REGION Network 53: Step[910] : Transfer PP Right X/Z-Axis Weight Check Pos
   RUNG wire#powerrail
      { S7_Templates := "SrcType := DInt" } EQ_Contact(in1 := "Unit1.Em5.ControlNodes".transferPnPRight.sequence.status.currentStep, in2 := #JOB_9_STEP_10)
      Contact( "Unit1.Em5.ControlNodes".transferPnPRight.sequence.status.seqActive )
      wire#w1
      I_Contact( "Unit1.Em5.ControlNodes".cm.softcam.transferPnPRightAxisX.pos04_weightCheck.inPos )
      wire#w2
      Coil( "Unit1.Em5.ControlNodes".transferPnPRight."step".action1[910] )
   END_RUNG
   RUNG wire#w1
      I_Contact( "Unit1.Em5.ControlNodes".cm.softcam.transferPnPRightAxisZ.pos04_weightCheck1.inPos )
   END_RUNG wire#w2
   RUNG wire#w1
      Contact( "Unit1.Em5.ControlNodes".cm.softcam.transferPnPRightAxisX.pos04_weightCheck.inPos )
      Contact( "Unit1.Em5.ControlNodes".cm.softcam.transferPnPRightAxisZ.pos04_weightCheck1.inPos )
      Coil( "Unit1.Em5.ControlNodes".transferPnPRight."step".transition1[910] )
   END_RUNG
   RUNG wire#w1
      Contact( "Unit1.Em5.ControlNodes".transferPnPRight."step".transition1[910] )
      { S7_Templates := "time_type := Time" } #statTonTime[910].TON(pt := T#100ms, et =>)
      Move(in := #JOB_9_STEP_30, out1 => "Unit1.Em5.ControlNodes".transferPnPRight.sequence.status.nextStep)
   END_RUNG
   // the same network as SCL:
   #_w1 := ("Unit1.Em5.ControlNodes".transferPnPRight.sequence.status.currentStep = #JOB_9_STEP_10) AND "Unit1.Em5.ControlNodes".transferPnPRight.sequence.status.seqActive;
   "Unit1.Em5.ControlNodes".transferPnPRight."step".action1[910] := #_w1 AND (NOT "Unit1.Em5.ControlNodes".cm.softcam.transferPnPRightAxisX.pos04_weightCheck.inPos OR NOT "Unit1.Em5.ControlNodes".cm.softcam.transferPnPRightAxisZ.pos04_weightCheck1.inPos);
   "Unit1.Em5.ControlNodes".transferPnPRight."step".transition1[910] := #_w1 AND "Unit1.Em5.ControlNodes".cm.softcam.transferPnPRightAxisX.pos04_weightCheck.inPos AND "Unit1.Em5.ControlNodes".cm.softcam.transferPnPRightAxisZ.pos04_weightCheck1.inPos;
   #statTonTime[910].TON(IN := #_w1 AND "Unit1.Em5.ControlNodes".transferPnPRight."step".transition1[910],
                         PT := T#100ms);
   IF #statTonTime[910].Q THEN
       "Unit1.Em5.ControlNodes".transferPnPRight.sequence.status.nextStep := #JOB_9_STEP_30;
   END_IF;
END_REGION

REGION Network 54: Step[930] : Transfer PP Right Y-Axis Weight Check Pos
   RUNG wire#powerrail
      { S7_Templates := "SrcType := DInt" } EQ_Contact(in1 := "Unit1.Em5.ControlNodes".transferPnPRight.sequence.status.currentStep, in2 := #JOB_9_STEP_30)
      Contact( "Unit1.Em5.ControlNodes".transferPnPRight.sequence.status.seqActive )
      wire#w1
      I_Contact( "Unit1.Em5.ControlNodes".cm.softcam.transferPnPRightAxisY.pos04_weightCheck.inPos )
      Coil( "Unit1.Em5.ControlNodes".transferPnPRight."step".action1[930] )
   END_RUNG
   RUNG wire#w1
      Contact( "Unit1.Em5.ControlNodes".cm.softcam.transferPnPRightAxisY.pos04_weightCheck.inPos )
      Coil( "Unit1.Em5.ControlNodes".transferPnPRight."step".transition1[930] )
   END_RUNG
   RUNG wire#w1
      Contact( "Unit1.Em5.ControlNodes".transferPnPRight."step".transition1[930] )
      { S7_Templates := "time_type := Time" } #statTonTime[930].TON(pt := T#100ms, et =>)
      Move(in := #JOB_9_STEP_31, out1 => "Unit1.Em5.ControlNodes".transferPnPRight.sequence.status.nextStep)
   END_RUNG
   // the same network as SCL:
   #_w1 := ("Unit1.Em5.ControlNodes".transferPnPRight.sequence.status.currentStep = #JOB_9_STEP_30) AND "Unit1.Em5.ControlNodes".transferPnPRight.sequence.status.seqActive;
   "Unit1.Em5.ControlNodes".transferPnPRight."step".action1[930] := #_w1 AND NOT "Unit1.Em5.ControlNodes".cm.softcam.transferPnPRightAxisY.pos04_weightCheck.inPos;
   "Unit1.Em5.ControlNodes".transferPnPRight."step".transition1[930] := #_w1 AND "Unit1.Em5.ControlNodes".cm.softcam.transferPnPRightAxisY.pos04_weightCheck.inPos;
   #statTonTime[930].TON(IN := #_w1 AND "Unit1.Em5.ControlNodes".transferPnPRight."step".transition1[930],
                         PT := T#100ms);
   IF #statTonTime[930].Q THEN
       "Unit1.Em5.ControlNodes".transferPnPRight.sequence.status.nextStep := #JOB_9_STEP_31;
   END_IF;
END_REGION

REGION Network 55: Step[931] : Transfer PP Right Z-Axis Weight Check Pos
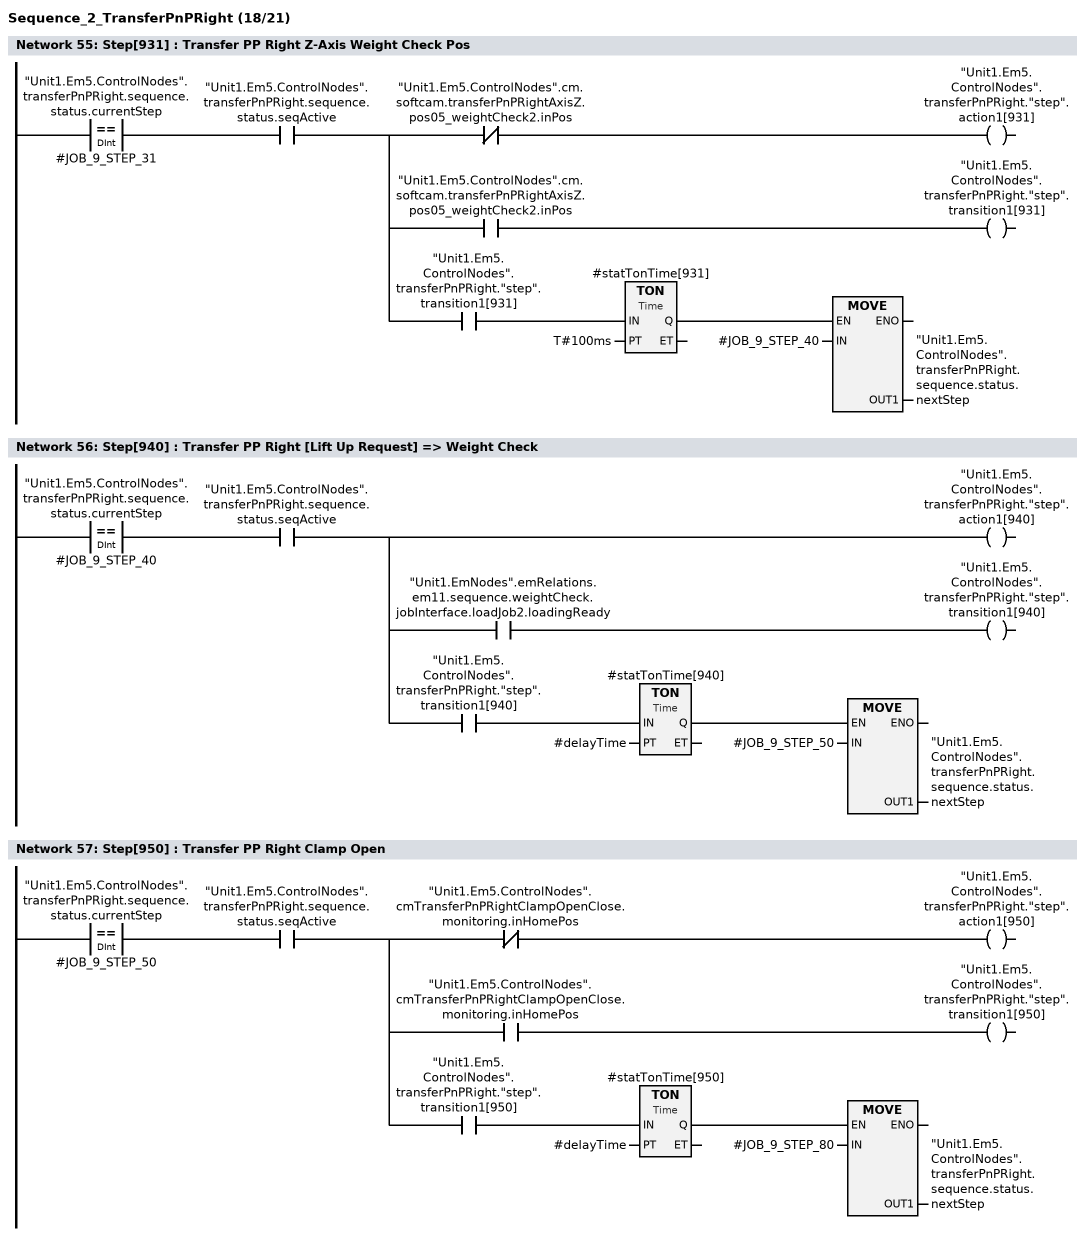
   RUNG wire#powerrail
      { S7_Templates := "SrcType := DInt" } EQ_Contact(in1 := "Unit1.Em5.ControlNodes".transferPnPRight.sequence.status.currentStep, in2 := #JOB_9_STEP_31)
      Contact( "Unit1.Em5.ControlNodes".transferPnPRight.sequence.status.seqActive )
      wire#w1
      I_Contact( "Unit1.Em5.ControlNodes".cm.softcam.transferPnPRightAxisZ.pos05_weightCheck2.inPos )
      Coil( "Unit1.Em5.ControlNodes".transferPnPRight."step".action1[931] )
   END_RUNG
   RUNG wire#w1
      Contact( "Unit1.Em5.ControlNodes".cm.softcam.transferPnPRightAxisZ.pos05_weightCheck2.inPos )
      Coil( "Unit1.Em5.ControlNodes".transferPnPRight."step".transition1[931] )
   END_RUNG
   RUNG wire#w1
      Contact( "Unit1.Em5.ControlNodes".transferPnPRight."step".transition1[931] )
      { S7_Templates := "time_type := Time" } #statTonTime[931].TON(pt := T#100ms, et =>)
      Move(in := #JOB_9_STEP_40, out1 => "Unit1.Em5.ControlNodes".transferPnPRight.sequence.status.nextStep)
   END_RUNG
   // the same network as SCL:
   #_w1 := ("Unit1.Em5.ControlNodes".transferPnPRight.sequence.status.currentStep = #JOB_9_STEP_31) AND "Unit1.Em5.ControlNodes".transferPnPRight.sequence.status.seqActive;
   "Unit1.Em5.ControlNodes".transferPnPRight."step".action1[931] := #_w1 AND NOT "Unit1.Em5.ControlNodes".cm.softcam.transferPnPRightAxisZ.pos05_weightCheck2.inPos;
   "Unit1.Em5.ControlNodes".transferPnPRight."step".transition1[931] := #_w1 AND "Unit1.Em5.ControlNodes".cm.softcam.transferPnPRightAxisZ.pos05_weightCheck2.inPos;
   #statTonTime[931].TON(IN := #_w1 AND "Unit1.Em5.ControlNodes".transferPnPRight."step".transition1[931],
                         PT := T#100ms);
   IF #statTonTime[931].Q THEN
       "Unit1.Em5.ControlNodes".transferPnPRight.sequence.status.nextStep := #JOB_9_STEP_40;
   END_IF;
END_REGION

REGION Network 56: Step[940] : Transfer PP Right [Lift Up Request] => Weight Check
   RUNG wire#powerrail
      { S7_Templates := "SrcType := DInt" } EQ_Contact(in1 := "Unit1.Em5.ControlNodes".transferPnPRight.sequence.status.currentStep, in2 := #JOB_9_STEP_40)
      Contact( "Unit1.Em5.ControlNodes".transferPnPRight.sequence.status.seqActive )
      wire#w1
      Coil( "Unit1.Em5.ControlNodes".transferPnPRight."step".action1[940] )
   END_RUNG
   RUNG wire#w1
      Contact( "Unit1.EmNodes".emRelations.em11.sequence.weightCheck.jobInterface.loadJob2.loadingReady )
      Coil( "Unit1.Em5.ControlNodes".transferPnPRight."step".transition1[940] )
   END_RUNG
   RUNG wire#w1
      Contact( "Unit1.Em5.ControlNodes".transferPnPRight."step".transition1[940] )
      { S7_Templates := "time_type := Time" } #statTonTime[940].TON(pt := #delayTime, et =>)
      Move(in := #JOB_9_STEP_50, out1 => "Unit1.Em5.ControlNodes".transferPnPRight.sequence.status.nextStep)
   END_RUNG
   // the same network as SCL:
   "Unit1.Em5.ControlNodes".transferPnPRight."step".action1[940] := ("Unit1.Em5.ControlNodes".transferPnPRight.sequence.status.currentStep = #JOB_9_STEP_40) AND "Unit1.Em5.ControlNodes".transferPnPRight.sequence.status.seqActive;
   "Unit1.Em5.ControlNodes".transferPnPRight."step".transition1[940] := ("Unit1.Em5.ControlNodes".transferPnPRight.sequence.status.currentStep = #JOB_9_STEP_40) AND "Unit1.Em5.ControlNodes".transferPnPRight.sequence.status.seqActive AND "Unit1.EmNodes".emRelations.em11.sequence.weightCheck.jobInterface.loadJob2.loadingReady;
   #statTonTime[940].TON(IN := ("Unit1.Em5.ControlNodes".transferPnPRight.sequence.status.currentStep = #JOB_9_STEP_40) AND "Unit1.Em5.ControlNodes".transferPnPRight.sequence.status.seqActive AND "Unit1.Em5.ControlNodes".transferPnPRight."step".transition1[940],
                         PT := #delayTime);
   IF #statTonTime[940].Q THEN
       "Unit1.Em5.ControlNodes".transferPnPRight.sequence.status.nextStep := #JOB_9_STEP_50;
   END_IF;
END_REGION

REGION Network 57: Step[950] : Transfer PP Right Clamp Open
   RUNG wire#powerrail
      { S7_Templates := "SrcType := DInt" } EQ_Contact(in1 := "Unit1.Em5.ControlNodes".transferPnPRight.sequence.status.currentStep, in2 := #JOB_9_STEP_50)
      Contact( "Unit1.Em5.ControlNodes".transferPnPRight.sequence.status.seqActive )
      wire#w1
      I_Contact( "Unit1.Em5.ControlNodes".cmTransferPnPRightClampOpenClose.monitoring.inHomePos )
      Coil( "Unit1.Em5.ControlNodes".transferPnPRight."step".action1[950] )
   END_RUNG
   RUNG wire#w1
      Contact( "Unit1.Em5.ControlNodes".cmTransferPnPRightClampOpenClose.monitoring.inHomePos )
      Coil( "Unit1.Em5.ControlNodes".transferPnPRight."step".transition1[950] )
   END_RUNG
   RUNG wire#w1
      Contact( "Unit1.Em5.ControlNodes".transferPnPRight."step".transition1[950] )
      { S7_Templates := "time_type := Time" } #statTonTime[950].TON(pt := #delayTime, et =>)
      Move(in := #JOB_9_STEP_80, out1 => "Unit1.Em5.ControlNodes".transferPnPRight.sequence.status.nextStep)
   END_RUNG
   // the same network as SCL:
   #_w1 := ("Unit1.Em5.ControlNodes".transferPnPRight.sequence.status.currentStep = #JOB_9_STEP_50) AND "Unit1.Em5.ControlNodes".transferPnPRight.sequence.status.seqActive;
   "Unit1.Em5.ControlNodes".transferPnPRight."step".action1[950] := #_w1 AND NOT "Unit1.Em5.ControlNodes".cmTransferPnPRightClampOpenClose.monitoring.inHomePos;
   "Unit1.Em5.ControlNodes".transferPnPRight."step".transition1[950] := #_w1 AND "Unit1.Em5.ControlNodes".cmTransferPnPRightClampOpenClose.monitoring.inHomePos;
   #statTonTime[950].TON(IN := #_w1 AND "Unit1.Em5.ControlNodes".transferPnPRight."step".transition1[950],
                         PT := #delayTime);
   IF #statTonTime[950].Q THEN
       "Unit1.Em5.ControlNodes".transferPnPRight.sequence.status.nextStep := #JOB_9_STEP_80;
   END_IF;
END_REGION

REGION Network 58: Step[980] : Transfer PP Right Y-Axis Wait Pos
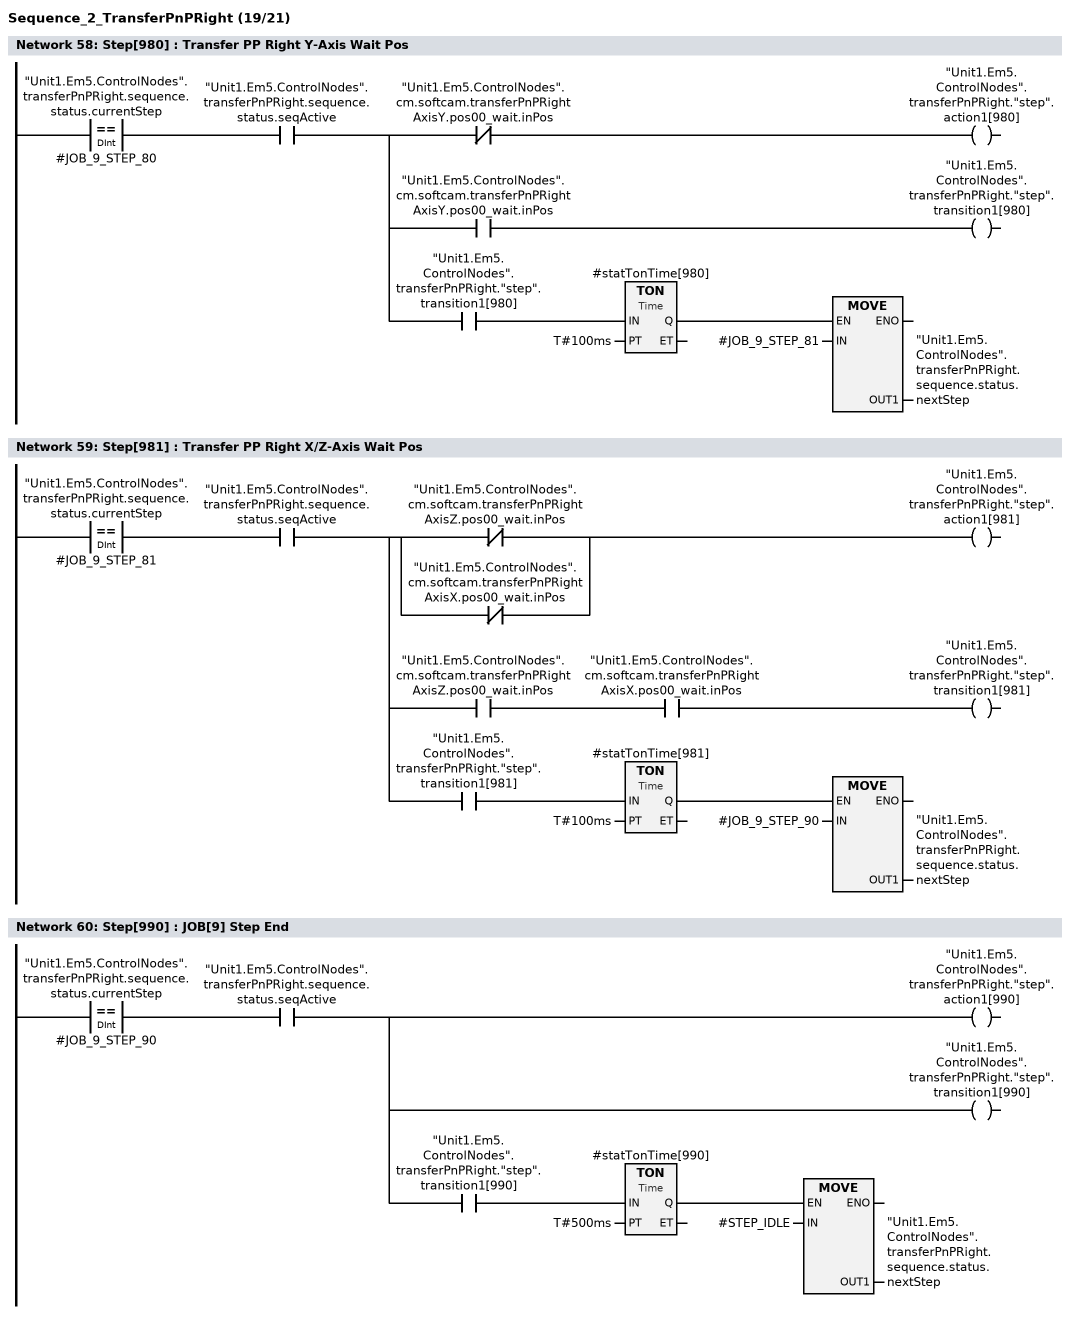
   RUNG wire#powerrail
      { S7_Templates := "SrcType := DInt" } EQ_Contact(in1 := "Unit1.Em5.ControlNodes".transferPnPRight.sequence.status.currentStep, in2 := #JOB_9_STEP_80)
      Contact( "Unit1.Em5.ControlNodes".transferPnPRight.sequence.status.seqActive )
      wire#w1
      I_Contact( "Unit1.Em5.ControlNodes".cm.softcam.transferPnPRightAxisY.pos00_wait.inPos )
      Coil( "Unit1.Em5.ControlNodes".transferPnPRight."step".action1[980] )
   END_RUNG
   RUNG wire#w1
      Contact( "Unit1.Em5.ControlNodes".cm.softcam.transferPnPRightAxisY.pos00_wait.inPos )
      Coil( "Unit1.Em5.ControlNodes".transferPnPRight."step".transition1[980] )
   END_RUNG
   RUNG wire#w1
      Contact( "Unit1.Em5.ControlNodes".transferPnPRight."step".transition1[980] )
      { S7_Templates := "time_type := Time" } #statTonTime[980].TON(pt := T#100ms, et =>)
      Move(in := #JOB_9_STEP_81, out1 => "Unit1.Em5.ControlNodes".transferPnPRight.sequence.status.nextStep)
   END_RUNG
   // the same network as SCL:
   #_w1 := ("Unit1.Em5.ControlNodes".transferPnPRight.sequence.status.currentStep = #JOB_9_STEP_80) AND "Unit1.Em5.ControlNodes".transferPnPRight.sequence.status.seqActive;
   "Unit1.Em5.ControlNodes".transferPnPRight."step".action1[980] := #_w1 AND NOT "Unit1.Em5.ControlNodes".cm.softcam.transferPnPRightAxisY.pos00_wait.inPos;
   "Unit1.Em5.ControlNodes".transferPnPRight."step".transition1[980] := #_w1 AND "Unit1.Em5.ControlNodes".cm.softcam.transferPnPRightAxisY.pos00_wait.inPos;
   #statTonTime[980].TON(IN := #_w1 AND "Unit1.Em5.ControlNodes".transferPnPRight."step".transition1[980],
                         PT := T#100ms);
   IF #statTonTime[980].Q THEN
       "Unit1.Em5.ControlNodes".transferPnPRight.sequence.status.nextStep := #JOB_9_STEP_81;
   END_IF;
END_REGION

REGION Network 59: Step[981] : Transfer PP Right X/Z-Axis Wait Pos
   RUNG wire#powerrail
      { S7_Templates := "SrcType := DInt" } EQ_Contact(in1 := "Unit1.Em5.ControlNodes".transferPnPRight.sequence.status.currentStep, in2 := #JOB_9_STEP_81)
      Contact( "Unit1.Em5.ControlNodes".transferPnPRight.sequence.status.seqActive )
      wire#w1
      I_Contact( "Unit1.Em5.ControlNodes".cm.softcam.transferPnPRightAxisZ.pos00_wait.inPos )
      wire#w2
      Coil( "Unit1.Em5.ControlNodes".transferPnPRight."step".action1[981] )
   END_RUNG
   RUNG wire#w1
      I_Contact( "Unit1.Em5.ControlNodes".cm.softcam.transferPnPRightAxisX.pos00_wait.inPos )
   END_RUNG wire#w2
   RUNG wire#w1
      Contact( "Unit1.Em5.ControlNodes".cm.softcam.transferPnPRightAxisZ.pos00_wait.inPos )
      Contact( "Unit1.Em5.ControlNodes".cm.softcam.transferPnPRightAxisX.pos00_wait.inPos )
      Coil( "Unit1.Em5.ControlNodes".transferPnPRight."step".transition1[981] )
   END_RUNG
   RUNG wire#w1
      Contact( "Unit1.Em5.ControlNodes".transferPnPRight."step".transition1[981] )
      { S7_Templates := "time_type := Time" } #statTonTime[981].TON(pt := T#100ms, et =>)
      Move(in := #JOB_9_STEP_90, out1 => "Unit1.Em5.ControlNodes".transferPnPRight.sequence.status.nextStep)
   END_RUNG
   // the same network as SCL:
   #_w1 := ("Unit1.Em5.ControlNodes".transferPnPRight.sequence.status.currentStep = #JOB_9_STEP_81) AND "Unit1.Em5.ControlNodes".transferPnPRight.sequence.status.seqActive;
   "Unit1.Em5.ControlNodes".transferPnPRight."step".action1[981] := #_w1 AND (NOT "Unit1.Em5.ControlNodes".cm.softcam.transferPnPRightAxisZ.pos00_wait.inPos OR NOT "Unit1.Em5.ControlNodes".cm.softcam.transferPnPRightAxisX.pos00_wait.inPos);
   "Unit1.Em5.ControlNodes".transferPnPRight."step".transition1[981] := #_w1 AND "Unit1.Em5.ControlNodes".cm.softcam.transferPnPRightAxisZ.pos00_wait.inPos AND "Unit1.Em5.ControlNodes".cm.softcam.transferPnPRightAxisX.pos00_wait.inPos;
   #statTonTime[981].TON(IN := #_w1 AND "Unit1.Em5.ControlNodes".transferPnPRight."step".transition1[981],
                         PT := T#100ms);
   IF #statTonTime[981].Q THEN
       "Unit1.Em5.ControlNodes".transferPnPRight.sequence.status.nextStep := #JOB_9_STEP_90;
   END_IF;
END_REGION

REGION Network 60: Step[990] : JOB[9] Step End
   RUNG wire#powerrail
      { S7_Templates := "SrcType := DInt" } EQ_Contact(in1 := "Unit1.Em5.ControlNodes".transferPnPRight.sequence.status.currentStep, in2 := #JOB_9_STEP_90)
      Contact( "Unit1.Em5.ControlNodes".transferPnPRight.sequence.status.seqActive )
      wire#w1
      Coil( "Unit1.Em5.ControlNodes".transferPnPRight."step".action1[990] )
   END_RUNG
   RUNG wire#w1
      Coil( "Unit1.Em5.ControlNodes".transferPnPRight."step".transition1[990] )
   END_RUNG
   RUNG wire#w1
      Contact( "Unit1.Em5.ControlNodes".transferPnPRight."step".transition1[990] )
      { S7_Templates := "time_type := Time" } #statTonTime[990].TON(pt := T#500ms, et =>)
      Move(in := #STEP_IDLE, out1 => "Unit1.Em5.ControlNodes".transferPnPRight.sequence.status.nextStep)
   END_RUNG
   // the same network as SCL:
   "Unit1.Em5.ControlNodes".transferPnPRight."step".action1[990] := ("Unit1.Em5.ControlNodes".transferPnPRight.sequence.status.currentStep = #JOB_9_STEP_90) AND "Unit1.Em5.ControlNodes".transferPnPRight.sequence.status.seqActive;
   "Unit1.Em5.ControlNodes".transferPnPRight."step".transition1[990] := ("Unit1.Em5.ControlNodes".transferPnPRight.sequence.status.currentStep = #JOB_9_STEP_90) AND "Unit1.Em5.ControlNodes".transferPnPRight.sequence.status.seqActive;
   #statTonTime[990].TON(IN := ("Unit1.Em5.ControlNodes".transferPnPRight.sequence.status.currentStep = #JOB_9_STEP_90) AND "Unit1.Em5.ControlNodes".transferPnPRight.sequence.status.seqActive AND "Unit1.Em5.ControlNodes".transferPnPRight."step".transition1[990],
                         PT := T#500ms);
   IF #statTonTime[990].Q THEN
       "Unit1.Em5.ControlNodes".transferPnPRight.sequence.status.nextStep := #STEP_IDLE;
   END_IF;
END_REGION

REGION Network 61: ******************** IMMEDIATE STOP *********************
END_REGION

REGION Network 62: Immediate Stop
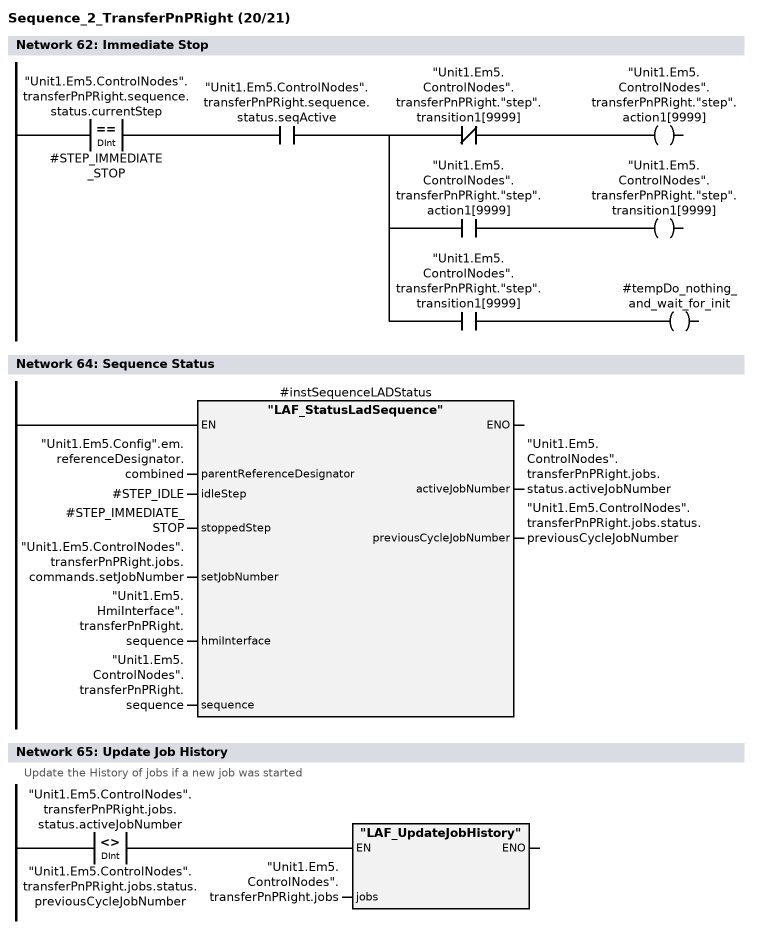
   RUNG wire#powerrail
      { S7_Templates := "SrcType := DInt" } EQ_Contact(in1 := "Unit1.Em5.ControlNodes".transferPnPRight.sequence.status.currentStep, in2 := #STEP_IMMEDIATE_STOP)
      Contact( "Unit1.Em5.ControlNodes".transferPnPRight.sequence.status.seqActive )
      wire#w1
      I_Contact( "Unit1.Em5.ControlNodes".transferPnPRight."step".transition1[9999] )
      Coil( "Unit1.Em5.ControlNodes".transferPnPRight."step".action1[9999] )
   END_RUNG
   RUNG wire#w1
      Contact( "Unit1.Em5.ControlNodes".transferPnPRight."step".action1[9999] )
      Coil( "Unit1.Em5.ControlNodes".transferPnPRight."step".transition1[9999] )
   END_RUNG
   RUNG wire#w1
      Contact( "Unit1.Em5.ControlNodes".transferPnPRight."step".transition1[9999] )
      Coil( #tempDo_nothing_and_wait_for_init )
   END_RUNG
   // the same network as SCL:
   #_w1 := ("Unit1.Em5.ControlNodes".transferPnPRight.sequence.status.currentStep = #STEP_IMMEDIATE_STOP) AND "Unit1.Em5.ControlNodes".transferPnPRight.sequence.status.seqActive;
   "Unit1.Em5.ControlNodes".transferPnPRight."step".action1[9999] := #_w1 AND NOT "Unit1.Em5.ControlNodes".transferPnPRight."step".transition1[9999];
   "Unit1.Em5.ControlNodes".transferPnPRight."step".transition1[9999] := #_w1 AND "Unit1.Em5.ControlNodes".transferPnPRight."step".action1[9999];
   #tempDo_nothing_and_wait_for_init := #_w1 AND "Unit1.Em5.ControlNodes".transferPnPRight."step".transition1[9999];
END_REGION

REGION Network 63: ********************** STATUS **************************
END_REGION

REGION Network 64: Sequence Status
   RUNG wire#powerrail
      #instSequenceLADStatus(parentReferenceDesignator := "Unit1.Em5.Config".em.referenceDesignator.combined, idleStep := #STEP_IDLE, stoppedStep := #STEP_IMMEDIATE_STOP, setJobNumber := "Unit1.Em5.ControlNodes".transferPnPRight.jobs.commands.setJobNumber, hmiInterface := "Unit1.Em5.HmiInterface".transferPnPRight.sequence, sequence := "Unit1.Em5.ControlNodes".transferPnPRight.sequence, activeJobNumber => "Unit1.Em5.ControlNodes".transferPnPRight.jobs.status.activeJobNumber, previousCycleJobNumber => "Unit1.Em5.ControlNodes".transferPnPRight.jobs.status.previousCycleJobNumber)
   END_RUNG
   // the same network as SCL:
   #instSequenceLADStatus(parentReferenceDesignator := "Unit1.Em5.Config".em.referenceDesignator.combined,   // "LAF_StatusLadSequence"
                          idleStep := #STEP_IDLE,
                          stoppedStep := #STEP_IMMEDIATE_STOP,
                          setJobNumber := "Unit1.Em5.ControlNodes".transferPnPRight.jobs.commands.setJobNumber,
                          hmiInterface := "Unit1.Em5.HmiInterface".transferPnPRight.sequence,
                          sequence := "Unit1.Em5.ControlNodes".transferPnPRight.sequence,
                          activeJobNumber => "Unit1.Em5.ControlNodes".transferPnPRight.jobs.status.activeJobNumber,
                          previousCycleJobNumber => "Unit1.Em5.ControlNodes".transferPnPRight.jobs.status.previousCycleJobNumber);
END_REGION

REGION Network 65: Update Job History
   // Update the History of jobs if a new job was started
   RUNG wire#powerrail
      { S7_Templates := "SrcType := DInt" } NE_Contact(in1 := "Unit1.Em5.ControlNodes".transferPnPRight.jobs.status.activeJobNumber, in2 := "Unit1.Em5.ControlNodes".transferPnPRight.jobs.status.previousCycleJobNumber)
      "LAF_UpdateJobHistory"(jobs := "Unit1.Em5.ControlNodes".transferPnPRight.jobs)
   END_RUNG
   // the same network as SCL:
   IF "Unit1.Em5.ControlNodes".transferPnPRight.jobs.status.activeJobNumber <> "Unit1.Em5.ControlNodes".transferPnPRight.jobs.status.previousCycleJobNumber THEN
       "LAF_UpdateJobHistory"(jobs := "Unit1.Em5.ControlNodes".transferPnPRight.jobs);
   END_IF;
END_REGION

REGION Network 66: Output Steps As String
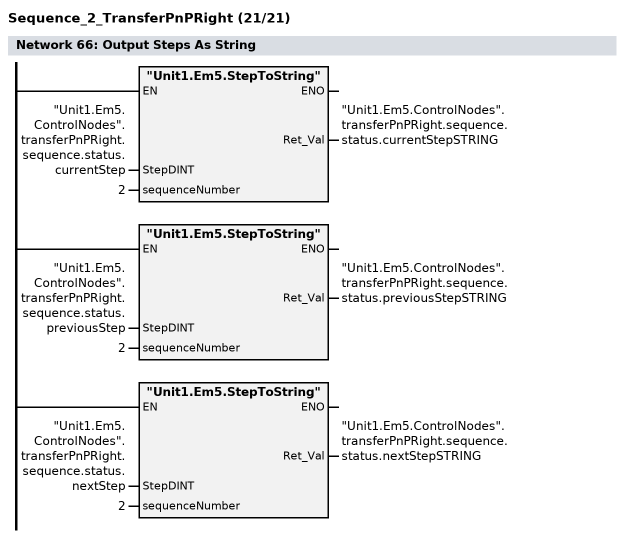
   RUNG wire#powerrail
      "Unit1.Em5.StepToString"(StepDINT := "Unit1.Em5.ControlNodes".transferPnPRight.sequence.status.currentStep, sequenceNumber := 2, Ret_Val => "Unit1.Em5.ControlNodes".transferPnPRight.sequence.status.currentStepSTRING)
   END_RUNG
   RUNG wire#powerrail
      "Unit1.Em5.StepToString"(StepDINT := "Unit1.Em5.ControlNodes".transferPnPRight.sequence.status.previousStep, sequenceNumber := 2, Ret_Val => "Unit1.Em5.ControlNodes".transferPnPRight.sequence.status.previousStepSTRING)
   END_RUNG
   RUNG wire#powerrail
      "Unit1.Em5.StepToString"(StepDINT := "Unit1.Em5.ControlNodes".transferPnPRight.sequence.status.nextStep, sequenceNumber := 2, Ret_Val => "Unit1.Em5.ControlNodes".transferPnPRight.sequence.status.nextStepSTRING)
   END_RUNG
   // the same network as SCL:
   "Unit1.Em5.ControlNodes".transferPnPRight.sequence.status.currentStepSTRING := "Unit1.Em5.StepToString"(StepDINT := "Unit1.Em5.ControlNodes".transferPnPRight.sequence.status.currentStep,
                           sequenceNumber := 2);
   "Unit1.Em5.ControlNodes".transferPnPRight.sequence.status.previousStepSTRING := "Unit1.Em5.StepToString"(StepDINT := "Unit1.Em5.ControlNodes".transferPnPRight.sequence.status.previousStep,
                           sequenceNumber := 2);
   "Unit1.Em5.ControlNodes".transferPnPRight.sequence.status.nextStepSTRING := "Unit1.Em5.StepToString"(StepDINT := "Unit1.Em5.ControlNodes".transferPnPRight.sequence.status.nextStep,
                           sequenceNumber := 2);
END_REGION
END_FUNCTION_BLOCK
